// TIA Portal project "Lab1" (V15)

(* hardware
DEVICE "S7-1200 station_1"  S7-1200 Station
   slot 0: "Rack_0"  S7-1200 Rack  Rack  V1.0
DEVICE "S7-1200 station_2"  S7-1200 Station
   slot 0: "Rack_0"  S7-1200 Rack  Rack  V1.0
DEVICE "S7-1200 station_3"  S7-1200 Station
   slot 0: "Rack_0"  S7-1200 Rack  Rack  V1.0
   slot 1: "PLC_1"  CPU 1214C AC/DC/Rly  6ES7 214-1BE30-0XB0  V2.2
*)

// ===== PLC "PLC_1"  CPU 1214C AC/DC/Rly =====

VAR_GLOBAL   // PLC tag table "Default tag table"
   "Start" AT %I0.1 : Bool;
   "Stop" AT %I0.5 : Bool;
   "KontaktorUkljucen" AT %I1.1 : Bool;
   "KontaktorSet" AT %Q0.2 : Bool;
   "MotorRadi" AT %I0.2 : Bool;
   "Auto" AT %I0.3 : Bool;
   "SigurnosniSklop" AT %I0.6 : Bool;
   "BiMetal" AT %I0.7 : Bool;
   "PrekoStrujna" AT %I1.0 : Bool;
   "Zelena" AT %Q0.0 : Bool;
   "Crvena" AT %Q0.1 : Bool;
   "MemBiMetal" AT %M0.0 : Bool;
   "MemPrekoStrujna" AT %M0.1 : Bool;
   "MemKontaktorGreska" AT %M0.2 : Bool;
   "MemSigurnosniSklop" AT %M0.3 : Bool;
   "MemGreskaGeneric" AT %M0.4 : Bool;
END_VAR

// folder: System blocks/Program resources

DATA_BLOCK "IEC_Timer_0_DB"   // DB1
{ S7_Optimized_Access := 'TRUE' }
AUTHOR : Simatic
FAMILY : IEC
NAME : IEC_TMR
VERSION : 1.0
// stored: InstanceOfName IEC_TIMER
"IEC_TIMER"
BEGIN
END_DATA_BLOCK

DATA_BLOCK "IEC_Timer_0_DB_1"   // DB2
{ S7_Optimized_Access := 'TRUE' }
AUTHOR : Simatic
FAMILY : IEC
NAME : IEC_TMR
VERSION : 1.0
// stored: InstanceOfName IEC_TIMER
"IEC_TIMER"
BEGIN
END_DATA_BLOCK

DATA_BLOCK "IEC_Timer_0_DB_2"   // DB3
{ S7_Optimized_Access := 'TRUE' }
AUTHOR : Simatic
FAMILY : IEC
NAME : IEC_TMR
VERSION : 1.0
// stored: InstanceOfName IEC_TIMER
"IEC_TIMER"
BEGIN
END_DATA_BLOCK

// folder: (top level)

ORGANIZATION_BLOCK "Main"   // OB1, LAD, ProgramCycle
TITLE = "Main Program Sweep (Cycle)"
{ S7_Optimized_Access := 'TRUE' }
VERSION : 0.1
BEGIN

REGION Network 1
   // Kada prekidac nije u auto rezimu, resetujemo greske i gasimo sve izlazne signale
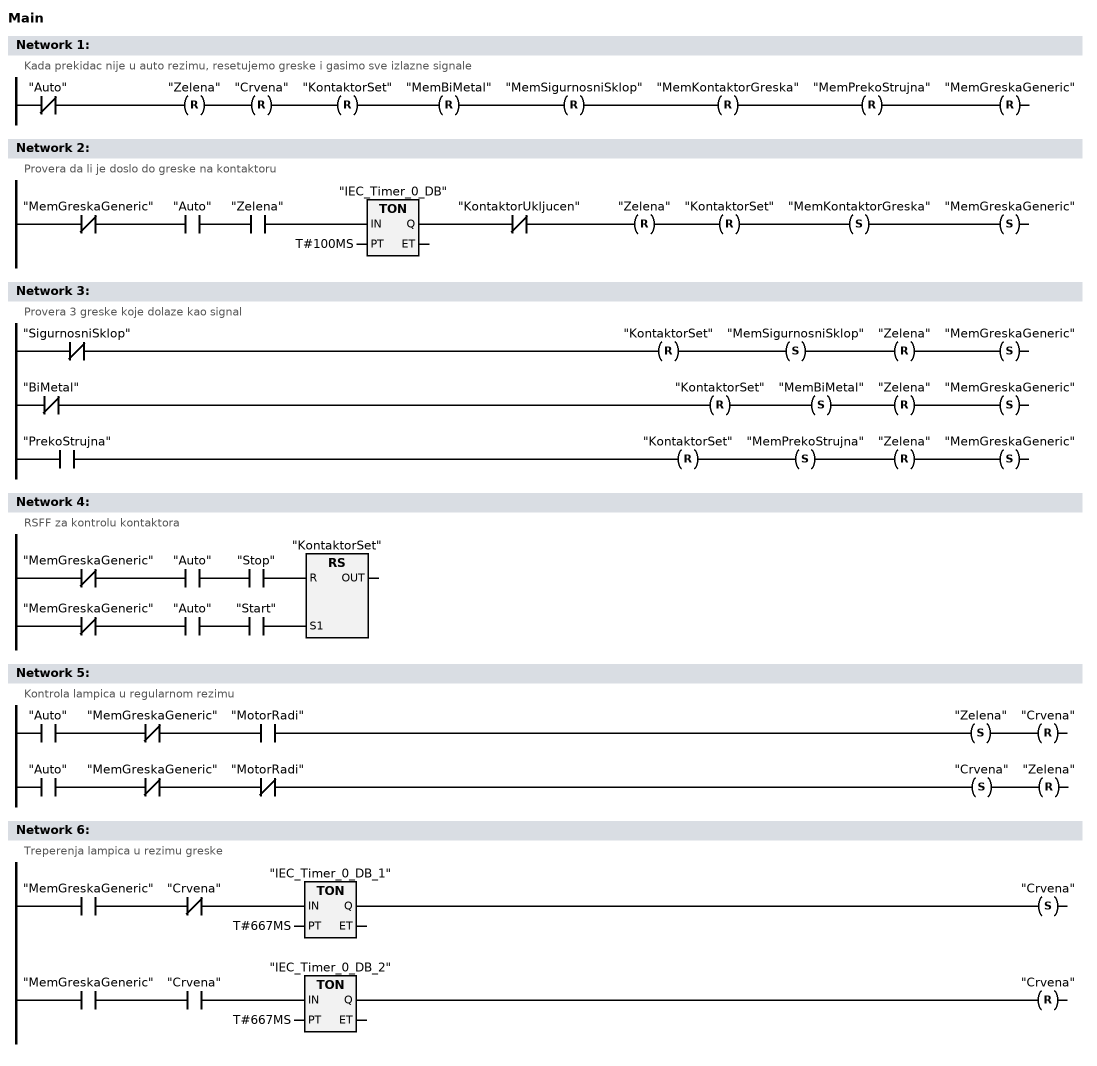
   RUNG wire#powerrail
      I_Contact( "Auto" )
      R_Coil( "Zelena" )
      R_Coil( "Crvena" )
      R_Coil( "KontaktorSet" )
      R_Coil( "MemBiMetal" )
      R_Coil( "MemSigurnosniSklop" )
      R_Coil( "MemKontaktorGreska" )
      R_Coil( "MemPrekoStrujna" )
      R_Coil( "MemGreskaGeneric" )
   END_RUNG
   // the same network as SCL:
   IF NOT "Auto" THEN
       "Zelena" := FALSE;
       "Crvena" := FALSE;
       "KontaktorSet" := FALSE;
       "MemBiMetal" := FALSE;
       "MemSigurnosniSklop" := FALSE;
       "MemKontaktorGreska" := FALSE;
       "MemPrekoStrujna" := FALSE;
       "MemGreskaGeneric" := FALSE;
   END_IF;
END_REGION

REGION Network 2
   // Provera da li je doslo do greske na kontaktoru
   "IEC_Timer_0_DB".TON(IN := NOT "MemGreskaGeneric" AND "Auto" AND "Zelena", PT := T#100MS);
   IF "IEC_Timer_0_DB".Q AND NOT "KontaktorUkljucen" THEN
       "Zelena" := FALSE;
       "KontaktorSet" := FALSE;
       "MemKontaktorGreska" := TRUE;
       "MemGreskaGeneric" := TRUE;
   END_IF;
END_REGION

REGION Network 3
   // Provera 3 greske koje dolaze kao signal
   RUNG wire#powerrail
      I_Contact( "SigurnosniSklop" )
      R_Coil( "KontaktorSet" )
      S_Coil( "MemSigurnosniSklop" )
      R_Coil( "Zelena" )
      S_Coil( "MemGreskaGeneric" )
   END_RUNG
   RUNG wire#powerrail
      I_Contact( "BiMetal" )
      R_Coil( "KontaktorSet" )
      S_Coil( "MemBiMetal" )
      R_Coil( "Zelena" )
      S_Coil( "MemGreskaGeneric" )
   END_RUNG
   RUNG wire#powerrail
      Contact( "PrekoStrujna" )
      R_Coil( "KontaktorSet" )
      S_Coil( "MemPrekoStrujna" )
      R_Coil( "Zelena" )
      S_Coil( "MemGreskaGeneric" )
   END_RUNG
   // the same network as SCL:
   IF NOT "SigurnosniSklop" THEN
       "KontaktorSet" := FALSE;
       "MemSigurnosniSklop" := TRUE;
       "Zelena" := FALSE;
       "MemGreskaGeneric" := TRUE;
   END_IF;
   IF NOT "BiMetal" THEN
       "KontaktorSet" := FALSE;
       "MemBiMetal" := TRUE;
       "Zelena" := FALSE;
       "MemGreskaGeneric" := TRUE;
   END_IF;
   IF "PrekoStrujna" THEN
       "KontaktorSet" := FALSE;
       "MemPrekoStrujna" := TRUE;
       "Zelena" := FALSE;
       "MemGreskaGeneric" := TRUE;
   END_IF;
END_REGION

REGION Network 4
   // RSFF za kontrolu kontaktora
   RUNG wire#powerrail
      I_Contact( "MemGreskaGeneric" )
      Contact( "Auto" )
      Contact( "Stop" )
      S_RS(operand := "KontaktorSet", s1 := wire#w1)
   END_RUNG
   RUNG wire#powerrail
      I_Contact( "MemGreskaGeneric" )
      Contact( "Auto" )
      Contact( "Start" )
   END_RUNG wire#w1
   // the same network as SCL:
   IF NOT "MemGreskaGeneric" AND "Auto" AND "Stop" THEN
       "KontaktorSet" := FALSE;   // RS flip-flop
   END_IF;
   IF NOT "MemGreskaGeneric" AND "Auto" AND "Start" THEN "KontaktorSet" := TRUE; END_IF;
END_REGION

REGION Network 5
   // Kontrola lampica u regularnom rezimu
   RUNG wire#powerrail
      Contact( "Auto" )
      I_Contact( "MemGreskaGeneric" )
      Contact( "MotorRadi" )
      S_Coil( "Zelena" )
      R_Coil( "Crvena" )
   END_RUNG
   RUNG wire#powerrail
      Contact( "Auto" )
      I_Contact( "MemGreskaGeneric" )
      I_Contact( "MotorRadi" )
      S_Coil( "Crvena" )
      R_Coil( "Zelena" )
   END_RUNG
   // the same network as SCL:
   IF "Auto" AND NOT "MemGreskaGeneric" AND "MotorRadi" THEN
       "Zelena" := TRUE;
       "Crvena" := FALSE;
   END_IF;
   IF "Auto" AND NOT "MemGreskaGeneric" AND NOT "MotorRadi" THEN
       "Crvena" := TRUE;
       "Zelena" := FALSE;
   END_IF;
END_REGION

REGION Network 6
   // Treperenja lampica u rezimu greske
   "IEC_Timer_0_DB_1".TON(IN := "MemGreskaGeneric" AND NOT "Crvena", PT := T#667MS);
   IF "IEC_Timer_0_DB_1".Q THEN "Crvena" := TRUE; END_IF;
   "IEC_Timer_0_DB_2".TON(IN := "MemGreskaGeneric" AND "Crvena", PT := T#667MS);
   IF "IEC_Timer_0_DB_2".Q THEN "Crvena" := FALSE; END_IF;
END_REGION
END_ORGANIZATION_BLOCK